// TIA Portal V16 export
// export: Created 2023-08-28T09:37:51.9348523Z, ExportSetting WithDefaults, DisplayName Totally Integrated Automation Portal, DisplayVersion V16 Update 6, DisplayName TIA Portal Version Control Interface, DisplayVersion V16 Update 2, DisplayName TIA Portal Openness, DisplayVersion V16 Update 6, DisplayName STEP 7 Professional, DisplayVersion V16 Update 6, DisplayName STEP 7 Safety, DisplayVersion V16, DisplayName WinCC Advanced, DisplayVersion V16 Update 6
DATA_BLOCK "dbdane"   // DB2
{ S7_Optimized_Access := 'FALSE' }
VERSION : 0.1
// stored: AutoNumber true, DBAccessibleFromOPCUA true, IsOnlyStoredInLoadMemory false, IsWriteProtectedInAS false
   VAR RETAIN
      TMR_ON_K3 : Time := T#10s;   // Wartość timera na dołączenie drugiej dodatkowej
      amplituda : Real := 95.0;   // Wiekośc zadana amplituda sygnału
      TMR_OFF_K3 : Time := T#10s;   // Wartość timera na odłączenie drugiej dodatkowej
      Manual_SV : Real;   // Wartość setpint zadana manualnie
      MV : Real;   // Wartość procentowa wyjącia regulatora PID [%]
      PV : Real;   // Wartość liczbowa sygnału analogowego cisnienia tłocznym
      tuning : Bool;
      zewnetrzne : Bool;
      dzialanie : Bool;
      Setpoint_SV : Real;   // Wartość zadanego ciśnienia do PID
      WYL : Bool;
      zerowanie : Bool;
      z_obiektu_analog : Word;
      do_obiektu_analog : Word;
      do_obiektu_pwm : Bool;
      PV_PER_B6 : Word;   // Ciśnienie tłoczny miasto strefa 2 (4-20mA)
      OUT_PER : Word;   // Sygnał wyjściowy Hz postać procesowa
      TMR_ON_K1 : Time;   // Wartość timera na dołączenie
      TMR_ON_K2 : Time;   // Wartość timera na dołączenie
      TMR_OFF_K1 : Time;   // Wartość timera na odłączenie
      TMR_OFF_K2 : Time;   // Wartość timera na odłączenie
      TMR_Hz : Time;   // Wartość timera na oczykiwanie 50Hz
      HMI : Struct
         PhysicalUnit : String[5] := '1/min';
         Output_PWM_USInt : USInt;
         ManualEnable_edge : Bool;
         ManualMode_visible : Bool;
         "sPid_Cmpt.b_Input_PER_On" : Bool;
         ErrorBits_Int : Int;
         ErrorAck_Int : Int;
         Warning_Int : Int;
         ErrorAck_Int_edge : Bool;
         ErrorAck : Bool;
         Acknowledge_visible : Bool;
         "sPid_Cmpt.r_Pv_Norm_OUT_2" : Real;   // Max wartośc procesowa przekazana z HMI
      END_STRUCT;
      OUT_PURE_Real : Real;   // Sygnał Hz w po scalowaniu do Hz
      Edge_1Hz_P1 : Bool;   // Pamięć zbocza naraztającego dla licznika pracy
      Edge_1Hz_P2 : Bool;   // Pamięć zbocza naraztającego dla licznika pracy
      Edge_1Hz_P3 : Bool;   // Pamięć zbocza naraztającego dla licznika pracy
      Edge_1Hz_P4 : Bool;
      "PID_Compact_1_sPid_Cmpt.r_Lmn_Hlm" : Real;
      "PID_Compact_1sPid_Cmpt.r_Pv_Norm_OUT_2" : Real;
      PID_Compact_1_ManualEnable : Bool;
      PID_Compact_1_ManualValue { ExternalWritable := 'False'} : Real;
      "PID_Compact_1_sPid_Cmpt.r_Lmn_Llm" : Real;
      "PID_Compact_1_sPid_Cmpt.r_Lmn_Pwm_PBTm" : Real;
      "PID_Compact_1_sPid_Cmpt.r_Lmn_Pwm_PPTm" : Real;
      "PID_Compact_1_sPid_Cmpt.r_Pv_HWrn" : Real;   // Nastawa progu ostrzerzenia PV wysoki
      "PID_Compact_1_sPid_Cmpt.r_Pv_LWrn" : Real;   // Nastawa progu ostrzerzenia PV niski
      "PID_Compact_1_sPid_Cmpt.r_Pv_Norm_IN_1" : Real;
      "PID_Compact_1_sPid_Cmpt.r_Pv_Norm_IN_2" : Real;
      "PID_Compact_1_sPid_Cmpt.r_Pv_Norm_OUT_1" : Real;
      "PID_Compact_1_sPid_Cmpt.r_Sp_Hlm" : Real;
      "PID_Compact_1_sPid_Cmpt.r_Sp_Llm" : Real;
      "PID_Compact_1_sPid_Cmpt.r_Pv_Hlm" : Real;
      "PID_Compact_1_sPid_Cmpt.r_Pv_Llm" : Real;
      Setpoint_bar_automat : Real;   // Zadana wartość ciśnienia w trybie automat (sterownik pobiera określoną wartośc zadaną w zależności od kierunku pompowania)
      PV_PER_B8 : Word;   // Ciśnienie ssanie suchobieg (4-20mA)
      MV_Real_b : Word;
      actPrzepływQ1_Real : Real;   // przepływ pompownia
      actPrzepływQ2_Real : Real;   // Zadane Hz pompomieszadło Word
      Switch_model_control_Tanks : Word;   // Sygnał sterowania zbiornikami -strategia
      Z11_Status : Word;
      Z12_Status : Word;
      Temp_SV : Word;   // Tymczasowa zadana wartość Hz
      Switch_model_control_P1P4 : Word;   // Sygnały sterowania strategią pompownia - 0= wyłaczone, 1=dosilanie, 2=przetłaczanie,3=automat, 4=ręczne
      tmp_Hz_ModeAlarm : Real;   // Przechwycone Hz podczas wystąpienia alarmu od max ciśnienie, prąd
      actPrzeoływQ1 { ExternalVisible := 'False'} : Int;   // Zmienna aktualny przepływ pompowia
      actPrzepływQ1_IA : Int := 0;   // Zmienna po konwersji do Integer
      Act_Value_B5_magistrala_bar : Real;   // Zmienna aktualnej wartości ciśnienia magistrala z PLC Zasuwy
      actHz_QW64 : Real := 0.0;   // Zmienna Hz pobrane z wyjacia analogowego
      actPrzepływQ1_IA_real : Real;   // aktualny przepływ Q1 pompownia z wyjścia analogowego
      PV_PER_B5 : Word;   // Ciśnienie magistrala strefa 1 (4-20mA)
      act_Value_B6 : Real;   // Ciśnienie tłoczny miasto strefa 2 (Real)
      act_Value_B5 : Real;   // Ciśnienie strefa 1 magistrala (Real)
      act_Value_B8 : Real;   // Ciśnienie ssania (Real)
      tmpdata_MV_PER : Word;   // Tymczasowa aktualnych Hz na potrzeby SCADA przekaznie między tymczasowym Hz a z regulatora PID
      tmpManualSV : LReal;   // pomocnicza przy konwersji wartość zadana manualnie SV
      ManualSV_Int : Int;   // wartość zadana manualnie SV (Word)
      tmpSV_manual_Hold : Int;   // tymczasowa wartość Hz w postaci procesowej podawana na wyjście w czasie podtrzymywania pompy wiodącej po odłaczeniu dodatkowej
      tmp_TR_ON_K1_1 : Int := 300;   // Zmienna czasu na dołączenie dodatkowej 1 pobierana przez algorytm PLC
      tmp_TR_ON_K2_1 : Int := 60;   // Zmienna czasu na dołączenie dodatkowej 2 pobierana przez algorytm PLC
      tmp_TR_OFF_K1_1 : Int := 5;   // Zmienna czasu na odołączenie dodatkowej 1 pobierana przez algorytm PLC
      tmp_TR_OFF_K2_1 : Int := 3;   // Zmienna czasu na odołączenie dodatkowej 2 pobierana przez algorytm PLC
      tmp_TR_50Hz_1 : Int := 15;   // Zmienna oczekiwania na 50Hz pobierana przez algorytm PLC
      tmp_TR_ON_K1_2 : Int := 30;   // Zmienna czasu na dołączenie dodatkowej 1 pobierana przez algorytm PLC
      tmp_TR_ON_K2_2 : Int := 30;   // Zmienna czasu na dołączenie dodatkowej 2 pobierana przez algorytm PLC
      tmp_TR_OFF_K1_2 : Int := 5;   // Zmienna czasu na odołączenie dodatkowej 1 pobierana przez algorytm PLC
      tmp_TR_OFF_K2_2 : Int := 5;   // Zmienna czasu na odołączenie dodatkowej 2 pobierana przez algorytm PLC
      tmp_TR_50Hz_2 : Int := 30;   // Zmienna oczekiwania na 50Hz pobierana przez algorytm PLC
      tmp_TR_ON_K1_3 : Int := 5;   // Zmienna czasu na dołączenie dodatkowej 1 pobierana przez algorytm PLC
      tmp_TR_ON_K2_3 : Int := 15;   // Zmienna czasu na dołączenie dodatkowej 2 pobierana przez algorytm PLC
      tmp_TR_OFF_K1_3 : Int := 2;   // Zmienna czasu na odołączenie dodatkowej 1 pobierana przez algorytm PLC
      tmp_TR_OFF_K2_3 : Int := 2;   // Zmienna czasu na odołączenie dodatkowej 2 pobierana przez algorytm PLC
      tmp_TR_50Hz_3 : Int := 5;   // Zmienna oczekiwania na 50Hz pobierana przez algorytm PLC
      tmpSV_spadekBar : Int;   // Hz tymczasowe dla spatku bar Max po odłączeniu dodatkowej
      Alarm_Max_bar : Real;   // Alarmowa wartość bar natychmiastowe wyłączenie układu
      tmpSV_spadek : Int := 15000;   // pomocnicza Hz tymczasowe dla opadającego ciśnienie z Max
      addressModbus_Fal : Byte;
      addressModbus_Q1_MPP04 : Byte;
      addressModbus_Q2_MPP04 : Byte;
      addressModbus_SlaveID : Byte;
      Wielkość_przeływu_Q1 : Real;
      Licznik_objętość_VF_Q1 : Real;
      Licznik_objętość_VR_Q1 : Real;
      Licznik_różnicowy_VD_Q1 : Real;
      Stan_licz_bjętości_GF_Q1 : Real;
      Stan_licz_rózicowego_obj_GD_Q1 : Real;
      _Stan_urządzenia_Q1 : Int;
      Wielkość_przeływu_Q2 : Real;
      Licznik_objętość_VF_Q2 : Real;
      Licznik_objętość_VR_Q2 : Real;
      Licznik_różnicowy_VD_Q2 : Real;
      Stan_licz_bjętości_GF_Q2 : Real;
      Stan_licz_rózicowego_obj_GD_Q2 : Real;
      _Stan_urządzenia_Q2 : Int;
      PV_analaog_B6 : Int;   // wartość analogowa z wejścia AI strafa 2
      PV_analaog_B7 : Int := 0;   // wartość analogowa z wejścia AI strafa 1
      PV_analaog_B8 : Int := 0;   // wartość analogowa z wejścia AI ssanie
      actSignalTank1 : Int;   // wartość analogowa procesowa poziom w zbiorniku 1
      actSignalTank2 : Int := 0;   // wartość analogowa procesowapoziom w zbiorniku 1
      actValu_Tank1 : Int;   // poziom w zbiorniku 1 po skalowaniu
      actValu_Tank2 : Int;   // poziom w zbiorniku 2 po skalowaniu
      actLevel_Tank1 : Int;   // poziom w zbiorniku 1 do SCADA
      actLevel_Tank2 : Int;   // poziom w zbiorniku 2 do SCADA
      actValu_Tank3 : Int;   // poziom w zbiorniku 3 po skalowaniu
      actLevel_Tank3 : Int;   // poziom w zbiorniku 3 do SCADA
      actSignalTank3 : Int;   // wartość analogowa procesowa poziom w zbiorniku 3
      ActivePump : Int;   // numer aktywnej pmpy - wiodącej 0=brak aktywnej
      pumpNum : Int;   // aktualnie sptawdzany licznik pompa
      chosenPump : Int;   // wybrana wiodąca pompa
   END_VAR
BEGIN
END_DATA_BLOCK
